TYPE ST_COM_SpeedControl :
STRUCT
	IMD_SpeedControl AT %Q*: ST_COM_IMD_SpdCntrl;
	SpeedControl_IMD AT %I*: ST_COM_SpdCntrl_IMD;
END_STRUCT
END_TYPE

(* stored: Version 1.1.0.1, ProductVersion 3.1.4020.12
   DUT ST_COM_SpeedControl: Id {115c4b03-7a6f-4488-ab83-16f25f78702c} *)
